# B&R Automation Studio project PLC code - cp (part 20)

#### Kernel2PLC_AutoCode.st
```iecst
// THIS CODE IS AUTOGENERATED. DO NOT MODIFY IT WITH AUTOMATION STUDIO
// Generation: 10/07/2024 16:17:34
// Program version: 2.1.4.0

ACTION Kernel2PLC_AutoCode:
gMachine.parSw.Clean.tiBetweenCleaningBlocks:=SECONDS_TO_TIME(HoldingRegister[3000]*1);
gMachine.parSw.Clean.iCleaningType:=HoldingRegister[3001];
gDing.parSw.rCalibrationValue:=INT_TO_REAL(HoldingRegister[3002])/10;
gMachine.parSw.Media.rThickness:=INT_TO_REAL(HoldingRegister[3003])/10;
gInks[1].parSw.NegPump.rLimitMeniscusDiffWarning:=INT_TO_REAL(HoldingRegister[3004])/10;
gInks[2].parSw.NegPump.rLimitMeniscusDiffWarning:=INT_TO_REAL(HoldingRegister[3005])/10;
gInks[3].parSw.NegPump.rLimitMeniscusDiffWarning:=INT_TO_REAL(HoldingRegister[3006])/10;
gInks[4].parSw.NegPump.rLimitMeniscusDiffWarning:=INT_TO_REAL(HoldingRegister[3007])/10;
gInks[5].parSw.NegPump.rLimitMeniscusDiffWarning:=INT_TO_REAL(HoldingRegister[3008])/10;
gInks[6].parSw.NegPump.rLimitMeniscusDiffWarning:=INT_TO_REAL(HoldingRegister[3009])/10;
gInks[7].parSw.NegPump.rLimitMeniscusDiffWarning:=INT_TO_REAL(HoldingRegister[3010])/10;
gInks[8].parSw.NegPump.rLimitMeniscusDiffWarning:=INT_TO_REAL(HoldingRegister[3011])/10;
gInks[9].parSw.NegPump.rLimitMeniscusDiffWarning:=INT_TO_REAL(HoldingRegister[3012])/10;
gInks[10].parSw.NegPump.rLimitMeniscusDiffWarning:=INT_TO_REAL(HoldingRegister[3013])/10;
gInks[11].parSw.NegPump.rLimitMeniscusDiffWarning:=INT_TO_REAL(HoldingRegister[3014])/10;
gInks[12].parSw.NegPump.rLimitMeniscusDiffWarning:=INT_TO_REAL(HoldingRegister[3015])/10;
gMachine.parSw.rMarginPrint:=INT_TO_REAL(HoldingRegister[3016])/10;
gMachine.parSw.Media.rWidth:=INT_TO_REAL(HoldingRegister[3017])/10;
gNonCrash[1].parSw.rGearBox:=INT_TO_REAL(HoldingRegister[3018])/1;
gNonCrash[1].parSw.rPerimeter:=INT_TO_REAL(HoldingRegister[3019])/10;
gNonCrash[1].parSw.rSpeedOffset:=INT_TO_REAL(HoldingRegister[3020])/10;
gMachine.parSw.rFirstHeadPosition:=INT_TO_REAL(HoldingRegister[3021])/1;
gMachine.parSw.rLastHeadPosition:=INT_TO_REAL(HoldingRegister[3022])/1;
gInks[1].parSw.PosPump.rSetPoint:=INT_TO_REAL(HoldingRegister[3023])/10;
gInks[2].parSw.PosPump.rSetPoint:=INT_TO_REAL(HoldingRegister[3024])/10;
gInks[3].parSw.PosPump.rSetPoint:=INT_TO_REAL(HoldingRegister[3025])/10;
gInks[4].parSw.PosPump.rSetPoint:=INT_TO_REAL(HoldingRegister[3026])/10;
gInks[5].parSw.PosPump.rSetPoint:=INT_TO_REAL(HoldingRegister[3027])/10;
gInks[6].parSw.PosPump.rSetPoint:=INT_TO_REAL(HoldingRegister[3028])/10;
gInks[7].parSw.PosPump.rSetPoint:=INT_TO_REAL(HoldingRegister[3029])/10;
gInks[8].parSw.PosPump.rSetPoint:=INT_TO_REAL(HoldingRegister[3030])/10;
gInks[9].parSw.PosPump.rSetPoint:=INT_TO_REAL(HoldingRegister[3031])/10;
gInks[10].parSw.PosPump.rSetPoint:=INT_TO_REAL(HoldingRegister[3032])/10;
gInks[11].parSw.PosPump.rSetPoint:=INT_TO_REAL(HoldingRegister[3033])/10;
gInks[12].parSw.PosPump.rSetPoint:=INT_TO_REAL(HoldingRegister[3034])/10;
gInks[1].parSw.NegPump.rSetPointMeniscus:=INT_TO_REAL(HoldingRegister[3035])/1;
gInks[2].parSw.NegPump.rSetPointMeniscus:=INT_TO_REAL(HoldingRegister[3036])/1;
gInks[3].parSw.NegPump.rSetPointMeniscus:=INT_TO_REAL(HoldingRegister[3037])/1;
gInks[4].parSw.NegPump.rSetPointMeniscus:=INT_TO_REAL(HoldingRegister[3038])/1;
gInks[5].parSw.NegPump.rSetPointMeniscus:=INT_TO_REAL(HoldingRegister[3039])/1;
gInks[6].parSw.NegPump.rSetPointMeniscus:=INT_TO_REAL(HoldingRegister[3040])/1;
gInks[7].parSw.NegPump.rSetPointMeniscus:=INT_TO_REAL(HoldingRegister[3041])/1;
gInks[8].parSw.NegPump.rSetPointMeniscus:=INT_TO_REAL(HoldingRegister[3042])/1;
gInks[9].parSw.NegPump.rSetPointMeniscus:=INT_TO_REAL(HoldingRegister[3043])/1;
gInks[10].parSw.NegPump.rSetPointMeniscus:=INT_TO_REAL(HoldingRegister[3044])/1;
gInks[11].parSw.NegPump.rSetPointMeniscus:=INT_TO_REAL(HoldingRegister[3045])/1;
gInks[12].parSw.NegPump.rSetPointMeniscus:=INT_TO_REAL(HoldingRegister[3046])/1;
gInks[1].parSw.Temp.rSetPointTemp:=INT_TO_REAL(HoldingRegister[3047])/10;
gInks[2].parSw.Temp.rSetPointTemp:=INT_TO_REAL(HoldingRegister[3048])/10;
gInks[3].parSw.Temp.rSetPointTemp:=INT_TO_REAL(HoldingRegister[3049])/10;
gInks[4].parSw.Temp.rSetPointTemp:=INT_TO_REAL(HoldingRegister[3050])/10;
gInks[5].parSw.Temp.rSetPointTemp:=INT_TO_REAL(HoldingRegister[3051])/10;
gInks[6].parSw.Temp.rSetPointTemp:=INT_TO_REAL(HoldingRegister[3052])/10;
gInks[7].parSw.Temp.rSetPointTemp:=INT_TO_REAL(HoldingRegister[3053])/10;
gInks[8].parSw.Temp.rSetPointTemp:=INT_TO_REAL(HoldingRegister[3054])/10;
gInks[9].parSw.Temp.rSetPointTemp:=INT_TO_REAL(HoldingRegister[3055])/10;
gInks[10].parSw.Temp.rSetPointTemp:=INT_TO_REAL(HoldingRegister[3056])/10;
gInks[11].parSw.Temp.rSetPointTemp:=INT_TO_REAL(HoldingRegister[3057])/10;
gInks[12].parSw.Temp.rSetPointTemp:=INT_TO_REAL(HoldingRegister[3058])/10;
gMachine.parSw.rBeltSpeedSetPoint:=INT_TO_REAL(HoldingRegister[3071])/10;
gInks[1].parSw.NegPump.rSetPointManual:=INT_TO_REAL(HoldingRegister[3072])/10;
gInks[2].parSw.NegPump.rSetPointManual:=INT_TO_REAL(HoldingRegister[3073])/10;
gInks[3].parSw.NegPump.rSetPointManual:=INT_TO_REAL(HoldingRegister[3074])/10;
gInks[4].parSw.NegPump.rSetPointManual:=INT_TO_REAL(HoldingRegister[3075])/10;
gInks[5].parSw.NegPump.rSetPointManual:=INT_TO_REAL(HoldingRegister[3076])/10;
gInks[6].parSw.NegPump.rSetPointManual:=INT_TO_REAL(HoldingRegister[3077])/10;
gInks[7].parSw.NegPump.rSetPointManual:=INT_TO_REAL(HoldingRegister[3078])/10;
gInks[8].parSw.NegPump.rSetPointManual:=INT_TO_REAL(HoldingRegister[3079])/10;
gInks[9].parSw.NegPump.rSetPointManual:=INT_TO_REAL(HoldingRegister[3080])/10;
gInks[10].parSw.NegPump.rSetPointManual:=INT_TO_REAL(HoldingRegister[3081])/10;
gInks[11].parSw.NegPump.rSetPointManual:=INT_TO_REAL(HoldingRegister[3082])/10;
gInks[12].parSw.NegPump.rSetPointManual:=INT_TO_REAL(HoldingRegister[3083])/10;
gInks[1].parSw.PosPump.rSetPointManual:=INT_TO_REAL(HoldingRegister[3084])/1;
gInks[2].parSw.PosPump.rSetPointManual:=INT_TO_REAL(HoldingRegister[3085])/1;
gInks[3].parSw.PosPump.rSetPointManual:=INT_TO_REAL(HoldingRegister[3086])/1;
gInks[4].parSw.PosPump.rSetPointManual:=INT_TO_REAL(HoldingRegister[3087])/1;
gInks[5].parSw.PosPump.rSetPointManual:=INT_TO_REAL(HoldingRegister[3088])/1;
gInks[6].parSw.PosPump.rSetPointManual:=INT_TO_REAL(HoldingRegister[3089])/1;
gInks[7].parSw.PosPump.rSetPointManual:=INT_TO_REAL(HoldingRegister[3090])/1;
gInks[8].parSw.PosPump.rSetPointManual:=INT_TO_REAL(HoldingRegister[3091])/1;
gInks[9].parSw.PosPump.rSetPointManual:=INT_TO_REAL(HoldingRegister[3092])/1;
gInks[10].parSw.PosPump.rSetPointManual:=INT_TO_REAL(HoldingRegister[3093])/1;
gInks[11].parSw.PosPump.rSetPointManual:=INT_TO_REAL(HoldingRegister[3094])/1;
gInks[12].parSw.PosPump.rSetPointManual:=INT_TO_REAL(HoldingRegister[3095])/1;
gMachine.parSw.tiDelayConsent:=SECONDS_TO_TIME(HoldingRegister[3096]*1);
gPhotoCells.parSw.rThicknessReference:=INT_TO_REAL(HoldingRegister[3097])/10;
gMachine.parSw.Clean.tiToCleanWhenPrinterStopped:=MINUTES_TO_TIME(HoldingRegister[3098]*1);
gTime.Params.UTCTimeZone:=HoldingRegister[3099];
gMachine.parSw.Clean.iCleanMotorSpeedFwd:=HoldingRegister[3100];
gMachine.parSw.Clean.iCleanMotorSpeedBwd:=HoldingRegister[3101];
ComandBool(In:=gMachine.parSw.Hw.xInstallnSensor,Com:=HoldingRegister[4000]);
ComandBool(In:=gTransVacuum[1].parSw.xActiveOutOfProduction,Com:=HoldingRegister[4001]);
ComandBool(In:=gTransVacuum[1].OrdersSw.xRunManual,Com:=HoldingRegister[4002]);
ComandBool(In:=gInks[1].parSw.xActTestMode,Com:=HoldingRegister[4003]);
ComandBool(In:=gInks[2].parSw.xActTestMode,Com:=HoldingRegister[4004]);
ComandBool(In:=gInks[3].parSw.xActTestMode,Com:=HoldingRegister[4005]);
ComandBool(In:=gInks[4].parSw.xActTestMode,Com:=HoldingRegister[4006]);
ComandBool(In:=gInks[5].parSw.xActTestMode,Com:=HoldingRegister[4007]);
ComandBool(In:=gInks[6].parSw.xActTestMode,Com:=HoldingRegister[4008]);
ComandBool(In:=gInks[7].parSw.xActTestMode,Com:=HoldingRegister[4009]);
ComandBool(In:=gInks[8].parSw.xActTestMode,Com:=HoldingRegister[4010]);
ComandBool(In:=gInks[9].parSw.xActTestMode,Com:=HoldingRegister[4011]);
ComandBool(In:=gInks[10].parSw.xActTestMode,Com:=HoldingRegister[4012]);
ComandBool(In:=gInks[11].parSw.xActTestMode,Com:=HoldingRegister[4013]);
ComandBool(In:=gInks[12].parSw.xActTestMode,Com:=HoldingRegister[4014]);
ComandBool(In:=gInks[1].parSw.xEnabledBarToPrint,Com:=HoldingRegister[4015]);
ComandBool(In:=gInks[2].parSw.xEnabledBarToPrint,Com:=HoldingRegister[4016]);
ComandBool(In:=gInks[3].parSw.xEnabledBarToPrint,Com:=HoldingRegister[4017]);
ComandBool(In:=gInks[4].parSw.xEnabledBarToPrint,Com:=HoldingRegister[4018]);
ComandBool(In:=gInks[5].parSw.xEnabledBarToPrint,Com:=HoldingRegister[4019]);
ComandBool(In:=gInks[6].parSw.xEnabledBarToPrint,Com:=HoldingRegister[4020]);
ComandBool(In:=gInks[7].parSw.xEnabledBarToPrint,Com:=HoldingRegister[4021]);
ComandBool(In:=gInks[8].parSw.xEnabledBarToPrint,Com:=HoldingRegister[4022]);
ComandBool(In:=gInks[9].parSw.xEnabledBarToPrint,Com:=HoldingRegister[4023]);
ComandBool(In:=gInks[10].parSw.xEnabledBarToPrint,Com:=HoldingRegister[4024]);
ComandBool(In:=gInks[11].parSw.xEnabledBarToPrint,Com:=HoldingRegister[4025]);
ComandBool(In:=gInks[12].parSw.xEnabledBarToPrint,Com:=HoldingRegister[4026]);
gTransVacuum[1].parSw.rVacPressureSetPointPerc:=INT_TO_REAL(HoldingRegister[4027])/10;
ComandBool(In:=gMachine.commandsSw.xToByPass_GI,Com:=HoldingRegister[4028]);
gMachine.parSw.Clean.iPiecesNumberToCleanL1:=HoldingRegister[4029];
gMachine.parSw.Clean.iPiecesNumberToCleanL2:=HoldingRegister[4030];
ComandBool(In:=gBlock[1].commands.xForceCleanNoDelay,Com:=HoldingRegister[4031]);
ComandBool(In:=gBlock[2].commands.xForceCleanNoDelay,Com:=HoldingRegister[4032]);
ComandBool(In:=gMachine.parSw.Clean.xCleaningBlocksInSeq,Com:=HoldingRegister[4033]);
gMachine.parSw.Safety.rMountedPieceOverthickness:=INT_TO_REAL(HoldingRegister[4036])/10;
ComandBool(In:=gMachine.parSw.Shot.xShotLine1,Com:=HoldingRegister[4038]);
ComandBool(In:=gMachine.parSw.Shot.xShotLine2,Com:=HoldingRegister[4039]);
ComandBool(In:=gMachine.parSw.Dtp.xDoubleLine,Com:=HoldingRegister[4040]);
gMachine.parSw.CleanBelt.tiCleaningBeltDuration:=SECONDS_TO_TIME(HoldingRegister[4041]*1);
gMachine.parSw.CleanBeltTop.tiCleaningBeltDuration:=SECONDS_TO_TIME(HoldingRegister[4042]*1);
ComandBool(In:=gBlock[1].commands.xEnableCleaningWithWater,Com:=HoldingRegister[4043]);
ComandBool(In:=gBlock[2].commands.xEnableCleaningWithWater,Com:=HoldingRegister[4044]);
ComandBool(In:=gMachine.parSw.xJamDetectEnable,Com:=HoldingRegister[4046]);
ComandBool(In:=gMachine.parSw.Clean.xEnableCleaningInStopMode,Com:=HoldingRegister[4047]);
ComandBool(In:=gBlock[1].parSw.xEnableToMovements,Com:=HoldingRegister[4048]);
ComandBool(In:=gBlock[2].parSw.xEnableToMovements,Com:=HoldingRegister[4049]);
ComandBool(In:=gNonCrash[1].parSw.xEnable,Com:=HoldingRegister[4050]);
ComandBool(In:=gInks[1].parSw.Temp.xTankHeaterEnabled,Com:=HoldingRegister[4051]);
ComandBool(In:=gInks[2].parSw.Temp.xTankHeaterEnabled,Com:=HoldingRegister[4052]);
ComandBool(In:=gInks[3].parSw.Temp.xTankHeaterEnabled,Com:=HoldingRegister[4053]);
ComandBool(In:=gInks[4].parSw.Temp.xTankHeaterEnabled,Com:=HoldingRegister[4054]);
ComandBool(In:=gInks[5].parSw.Temp.xTankHeaterEnabled,Com:=HoldingRegister[4055]);
ComandBool(In:=gInks[6].parSw.Temp.xTankHeaterEnabled,Com:=HoldingRegister[4056]);
ComandBool(In:=gInks[7].parSw.Temp.xTankHeaterEnabled,Com:=HoldingRegister[4057]);
ComandBool(In:=gInks[8].parSw.Temp.xTankHeaterEnabled,Com:=HoldingRegister[4058]);
ComandBool(In:=gInks[9].parSw.Temp.xTankHeaterEnabled,Com:=HoldingRegister[4059]);
ComandBool(In:=gInks[10].parSw.Temp.xTankHeaterEnabled,Com:=HoldingRegister[4060]);
ComandBool(In:=gInks[11].parSw.Temp.xTankHeaterEnabled,Com:=HoldingRegister[4061]);
ComandBool(In:=gInks[12].parSw.Temp.xTankHeaterEnabled,Com:=HoldingRegister[4062]);
ComandBool(In:=gBlock[1].parSw.xEnableToPrint,Com:=HoldingRegister[4063]);
ComandBool(In:=gBlock[2].parSw.xEnableToPrint,Com:=HoldingRegister[4064]);
ComandBool(In:=gMachine.parSw.Electronics.xPrintServerOK,Com:=HoldingRegister[4065]);
ComandBool(In:=gMachine.parSw.Electronics.xRobotReadyL1,Com:=HoldingRegister[4066]);
ComandBool(In:=gMachine.parSw.Electronics.xRobotReadyL2,Com:=HoldingRegister[4067]);
ComandBool(In:=gMachine.parSw.PCs.xExistPC1,Com:=HoldingRegister[4068]);
ComandBool(In:=gMachine.parSw.PCs.xExistPC2,Com:=HoldingRegister[4069]);
gMachine.parSw.iFaultComPcPlc:=HoldingRegister[4070];
ComandBool(In:=gBlock[1].commands.xForceCleanDelay,Com:=HoldingRegister[4073]);
ComandBool(In:=gBlock[2].commands.xForceCleanDelay,Com:=HoldingRegister[4074]);
ComandBool(In:=gBlock[1].commands.xToCleanPosition,Com:=HoldingRegister[4075]);
ComandBool(In:=gBlock[2].commands.xToCleanPosition,Com:=HoldingRegister[4076]);
ComandBool(In:=gMachine.parSw.CleanBelt.xCleanBeltByTiles,Com:=HoldingRegister[4077]);
ComandBool(In:=gMachine.parSw.CleanBelt.xCleanBeltByTime,Com:=HoldingRegister[4078]);
ComandBool(In:=gMachine.parSw.CleanBeltTop.xCleanBeltByTiles,Com:=HoldingRegister[4079]);
ComandBool(In:=gMachine.parSw.CleanBeltTop.xCleanBeltByTime,Com:=HoldingRegister[4080]);
ComandBool(In:=gBlock[1].commands.Manual.xManIclaBack,Com:=HoldingRegister[4081]);
ComandBool(In:=gBlock[2].commands.Manual.xManIclaBack,Com:=HoldingRegister[4082]);
ComandBool(In:=gBlock[1].commands.Manual.xManBarsDown,Com:=HoldingRegister[4083]);
ComandBool(In:=gBlock[2].commands.Manual.xManBarsDown,Com:=HoldingRegister[4084]);
ComandBool(In:=gBlock[1].commands.Manual.xManIclaForward,Com:=HoldingRegister[4085]);
ComandBool(In:=gBlock[2].commands.Manual.xManIclaForward,Com:=HoldingRegister[4086]);
gInks[1].parSw.iInkConsumption:=HoldingRegister[4087];
gInks[2].parSw.iInkConsumption:=HoldingRegister[4088];
gInks[3].parSw.iInkConsumption:=HoldingRegister[4089];
gInks[4].parSw.iInkConsumption:=HoldingRegister[4090];
gInks[5].parSw.iInkConsumption:=HoldingRegister[4091];
gInks[6].parSw.iInkConsumption:=HoldingRegister[4092];
gInks[7].parSw.iInkConsumption:=HoldingRegister[4093];
gInks[8].parSw.iInkConsumption:=HoldingRegister[4094];
gInks[9].parSw.iInkConsumption:=HoldingRegister[4095];
gInks[10].parSw.iInkConsumption:=HoldingRegister[4096];
gInks[11].parSw.iInkConsumption:=HoldingRegister[4097];
gInks[12].parSw.iInkConsumption:=HoldingRegister[4098];
ComandBool(In:=gInks[1].parSw.xReverseOnManual,Com:=HoldingRegister[4099]);
ComandBool(In:=gInks[2].parSw.xReverseOnManual,Com:=HoldingRegister[4100]);
ComandBool(In:=gInks[3].parSw.xReverseOnManual,Com:=HoldingRegister[4101]);
ComandBool(In:=gInks[4].parSw.xReverseOnManual,Com:=HoldingRegister[4102]);
ComandBool(In:=gInks[5].parSw.xReverseOnManual,Com:=HoldingRegister[4103]);
ComandBool(In:=gInks[6].parSw.xReverseOnManual,Com:=HoldingRegister[4104]);
ComandBool(In:=gInks[7].parSw.xReverseOnManual,Com:=HoldingRegister[4105]);
ComandBool(In:=gInks[8].parSw.xReverseOnManual,Com:=HoldingRegister[4106]);
ComandBool(In:=gInks[9].parSw.xReverseOnManual,Com:=HoldingRegister[4107]);
ComandBool(In:=gInks[10].parSw.xReverseOnManual,Com:=HoldingRegister[4108]);
ComandBool(In:=gInks[11].parSw.xReverseOnManual,Com:=HoldingRegister[4109]);
ComandBool(In:=gInks[12].parSw.xReverseOnManual,Com:=HoldingRegister[4110]);
gInks[1].parSw.Config.iInkType:=HoldingRegister[4111];
gInks[2].parSw.Config.iInkType:=HoldingRegister[4112];
gInks[3].parSw.Config.iInkType:=HoldingRegister[4113];
gInks[4].parSw.Config.iInkType:=HoldingRegister[4114];
gInks[5].parSw.Config.iInkType:=HoldingRegister[4115];
gInks[6].parSw.Config.iInkType:=HoldingRegister[4116];
gInks[7].parSw.Config.iInkType:=HoldingRegister[4117];
gInks[8].parSw.Config.iInkType:=HoldingRegister[4118];
gInks[9].parSw.Config.iInkType:=HoldingRegister[4119];
gInks[10].parSw.Config.iInkType:=HoldingRegister[4120];
gInks[11].parSw.Config.iInkType:=HoldingRegister[4121];
gInks[12].parSw.Config.iInkType:=HoldingRegister[4122];
ComandBool(In:=gMachine.commandsSw.xStart_GI,Com:=HoldingRegister[4123]);
ComandBool(In:=gMachine.commandsSw.xStop_GI,Com:=HoldingRegister[4124]);
ComandBool(In:=gMachine.commandsSw.xPause_GI,Com:=HoldingRegister[4125]);
ComandBool(In:=gMachine.commands.xCompenserLine1,Com:=HoldingRegister[4126]);
ComandBool(In:=gMachine.commands.xCompenserLine2,Com:=HoldingRegister[4127]);
ComandBool(In:=gBlock[1].commands.Manual.xManBarsUp,Com:=HoldingRegister[4128]);
ComandBool(In:=gBlock[2].commands.Manual.xManBarsUp,Com:=HoldingRegister[4129]);
ComandBool(In:=gBlock[1].commands.xIclaHomeOrderInterrupt,Com:=HoldingRegister[4130]);
ComandBool(In:=gBlock[2].commands.xIclaHomeOrderInterrupt,Com:=HoldingRegister[4131]);
ComandBool(In:=gMachine.parSw.Electronics.xIsPBF,Com:=HoldingRegister[4132]);
ComandBool(In:=gMachine.commandsSw.xToLaboratory_GI,Com:=HoldingRegister[4133]);
gMachine.parSw.CleanBelt.iSPTilesToCleanBelt:=HoldingRegister[4134];
ComandBool(In:=gMachine.parSw.CleanBelt.xCleanBeltContinue,Com:=HoldingRegister[4135]);
gMachine.parSw.CleanBeltTop.iSPTilesToCleanBelt:=HoldingRegister[4136];
ComandBool(In:=gMachine.parSw.CleanBeltTop.xCleanBeltContinue,Com:=HoldingRegister[4137]);
ComandBool(In:=gInks[1].ordersSw.xStartManual,Com:=HoldingRegister[4138]);
ComandBool(In:=gInks[2].ordersSw.xStartManual,Com:=HoldingRegister[4139]);
ComandBool(In:=gInks[3].ordersSw.xStartManual,Com:=HoldingRegister[4140]);
ComandBool(In:=gInks[4].ordersSw.xStartManual,Com:=HoldingRegister[4141]);
ComandBool(In:=gInks[5].ordersSw.xStartManual,Com:=HoldingRegister[4142]);
ComandBool(In:=gInks[6].ordersSw.xStartManual,Com:=HoldingRegister[4143]);
ComandBool(In:=gInks[7].ordersSw.xStartManual,Com:=HoldingRegister[4144]);
ComandBool(In:=gInks[8].ordersSw.xStartManual,Com:=HoldingRegister[4145]);
ComandBool(In:=gInks[9].ordersSw.xStartManual,Com:=HoldingRegister[4146]);
ComandBool(In:=gInks[10].ordersSw.xStartManual,Com:=HoldingRegister[4147]);
ComandBool(In:=gInks[11].ordersSw.xStartManual,Com:=HoldingRegister[4148]);
ComandBool(In:=gInks[12].ordersSw.xStartManual,Com:=HoldingRegister[4149]);
ComandBool(In:=gMachine.parSw.CleanBelt.xCleanBeltForced,Com:=HoldingRegister[4150]);
ComandBool(In:=gMachine.parSw.CleanBeltTop.xCleanBeltForced,Com:=HoldingRegister[4151]);
ComandBool(In:=gMachine.parSw.Clean.xCleanSystemByPieces,Com:=HoldingRegister[4152]);
ComandBool(In:=gMachine.parSw.Clean.xCleanSystemByTime,Com:=HoldingRegister[4153]);
ComandBool(In:=gBlock[1].commands.Manual.xManTrayIn,Com:=HoldingRegister[4154]);
ComandBool(In:=gBlock[2].commands.Manual.xManTrayIn,Com:=HoldingRegister[4155]);
ComandBool(In:=gBlock[1].commands.Manual.xManTrayOut,Com:=HoldingRegister[4156]);
ComandBool(In:=gBlock[2].commands.Manual.xManTrayOut,Com:=HoldingRegister[4157]);
ComandBool(In:=gMachine.parSw.xMachineDirection,Com:=HoldingRegister[4159]);
ComandBool(In:=gMachine.parSw.PCs.xKeepPcsOn,Com:=HoldingRegister[4161]);
gTransVacuum[1].parSw.rManSetPoint:=INT_TO_REAL(HoldingRegister[4162])/10;
ComandBool(In:=gBlock[1].commands.Manual.xManVenturi,Com:=HoldingRegister[4163]);
ComandBool(In:=gBlock[2].commands.Manual.xManVenturi,Com:=HoldingRegister[4164]);
gInks[1].parSw.Config.iMappingBar:=HoldingRegister[4165];
gInks[2].parSw.Config.iMappingBar:=HoldingRegister[4166];
gInks[3].parSw.Config.iMappingBar:=HoldingRegister[4167];
gInks[4].parSw.Config.iMappingBar:=HoldingRegister[4168];
gInks[5].parSw.Config.iMappingBar:=HoldingRegister[4169];
gInks[6].parSw.Config.iMappingBar:=HoldingRegister[4170];
gInks[7].parSw.Config.iMappingBar:=HoldingRegister[4171];
gInks[8].parSw.Config.iMappingBar:=HoldingRegister[4172];
gInks[9].parSw.Config.iMappingBar:=HoldingRegister[4173];
gInks[10].parSw.Config.iMappingBar:=HoldingRegister[4174];
gInks[11].parSw.Config.iMappingBar:=HoldingRegister[4175];
gInks[12].parSw.Config.iMappingBar:=HoldingRegister[4176];
ComandBool(In:=gInks[1].ordersSw.xStartInks,Com:=HoldingRegister[4177]);
ComandBool(In:=gInks[2].ordersSw.xStartInks,Com:=HoldingRegister[4178]);
ComandBool(In:=gInks[3].ordersSw.xStartInks,Com:=HoldingRegister[4179]);
ComandBool(In:=gInks[4].ordersSw.xStartInks,Com:=HoldingRegister[4180]);
ComandBool(In:=gInks[5].ordersSw.xStartInks,Com:=HoldingRegister[4181]);
ComandBool(In:=gInks[6].ordersSw.xStartInks,Com:=HoldingRegister[4182]);
ComandBool(In:=gInks[7].ordersSw.xStartInks,Com:=HoldingRegister[4183]);
ComandBool(In:=gInks[8].ordersSw.xStartInks,Com:=HoldingRegister[4184]);
ComandBool(In:=gInks[9].ordersSw.xStartInks,Com:=HoldingRegister[4185]);
ComandBool(In:=gInks[10].ordersSw.xStartInks,Com:=HoldingRegister[4186]);
ComandBool(In:=gInks[11].ordersSw.xStartInks,Com:=HoldingRegister[4187]);
ComandBool(In:=gInks[12].ordersSw.xStartInks,Com:=HoldingRegister[4188]);
gMachine.parSw.Safety.rMarginSafePrint:=INT_TO_REAL(HoldingRegister[4189])/10;
gMachine.parSw.Media.rLength:=INT_TO_REAL(HoldingRegister[4190])/10;
gBelt.parSw.rAxisLength:=INT_TO_REAL(HoldingRegister[4191])/10;
gMachine.parSw.Dtp.iModeLine1:=HoldingRegister[4192];
gMachine.parSw.Dtp.iModeLine2:=HoldingRegister[4193];
gMachine.parSw.Suction.iBlowerMode:=HoldingRegister[4194];
ComandBool(In:=gMachine.commandsSw.xToNormal_GI,Com:=HoldingRegister[4195]);
gBlock[1].parSw.rOffsetCleanMtrAdjust:=INT_TO_REAL(HoldingRegister[4196])/10;
gBlock[2].parSw.rOffsetCleanMtrAdjust:=INT_TO_REAL(HoldingRegister[4197])/10;
gBlock[1].parSw.rOffsetCleanMtrOperatr:=INT_TO_REAL(HoldingRegister[4198])/10;
gBlock[2].parSw.rOffsetCleanMtrOperatr:=INT_TO_REAL(HoldingRegister[4199])/10;
ComandBool(In:=gInks[1].parSw.xOnReverseCapped,Com:=HoldingRegister[4200]);
ComandBool(In:=gInks[2].parSw.xOnReverseCapped,Com:=HoldingRegister[4201]);
ComandBool(In:=gInks[3].parSw.xOnReverseCapped,Com:=HoldingRegister[4202]);
ComandBool(In:=gInks[4].parSw.xOnReverseCapped,Com:=HoldingRegister[4203]);
ComandBool(In:=gInks[5].parSw.xOnReverseCapped,Com:=HoldingRegister[4204]);
ComandBool(In:=gInks[6].parSw.xOnReverseCapped,Com:=HoldingRegister[4205]);
ComandBool(In:=gInks[7].parSw.xOnReverseCapped,Com:=HoldingRegister[4206]);
ComandBool(In:=gInks[8].parSw.xOnReverseCapped,Com:=HoldingRegister[4207]);
ComandBool(In:=gInks[9].parSw.xOnReverseCapped,Com:=HoldingRegister[4208]);
ComandBool(In:=gInks[10].parSw.xOnReverseCapped,Com:=HoldingRegister[4209]);
ComandBool(In:=gInks[11].parSw.xOnReverseCapped,Com:=HoldingRegister[4210]);
ComandBool(In:=gInks[12].parSw.xOnReverseCapped,Com:=HoldingRegister[4211]);
ComandBool(In:=gInks[1].parSw.xOnReverseCleaning,Com:=HoldingRegister[4212]);
ComandBool(In:=gInks[2].parSw.xOnReverseCleaning,Com:=HoldingRegister[4213]);
ComandBool(In:=gInks[3].parSw.xOnReverseCleaning,Com:=HoldingRegister[4214]);
ComandBool(In:=gInks[4].parSw.xOnReverseCleaning,Com:=HoldingRegister[4215]);
ComandBool(In:=gInks[5].parSw.xOnReverseCleaning,Com:=HoldingRegister[4216]);
ComandBool(In:=gInks[6].parSw.xOnReverseCleaning,Com:=HoldingRegister[4217]);
ComandBool(In:=gInks[7].parSw.xOnReverseCleaning,Com:=HoldingRegister[4218]);
ComandBool(In:=gInks[8].parSw.xOnReverseCleaning,Com:=HoldingRegister[4219]);
ComandBool(In:=gInks[9].parSw.xOnReverseCleaning,Com:=HoldingRegister[4220]);
ComandBool(In:=gInks[10].parSw.xOnReverseCleaning,Com:=HoldingRegister[4221]);
ComandBool(In:=gInks[11].parSw.xOnReverseCleaning,Com:=HoldingRegister[4222]);
ComandBool(In:=gInks[12].parSw.xOnReverseCleaning,Com:=HoldingRegister[4223]);
ComandBool(In:=gMachine.commands.xAllToCap,Com:=HoldingRegister[4224]);
ComandBool(In:=gMachine.commands.xAllToPrint,Com:=HoldingRegister[4225]);
ComandBool(In:=gPhotoCells.ordersSw.xMoveDown,Com:=HoldingRegister[4226]);
gPhotoCells.parSw.rMechOffset:=INT_TO_REAL(HoldingRegister[4227])/10;
ComandBool(In:=gPhotoCells.ordersSw.xMoveUp,Com:=HoldingRegister[4228]);
ComandBool(In:=gInks[1].ordersSw.xPowPrintHead,Com:=HoldingRegister[4229]);
ComandBool(In:=gInks[2].ordersSw.xPowPrintHead,Com:=HoldingRegister[4230]);
ComandBool(In:=gInks[3].ordersSw.xPowPrintHead,Com:=HoldingRegister[4231]);
ComandBool(In:=gInks[4].ordersSw.xPowPrintHead,Com:=HoldingRegister[4232]);
ComandBool(In:=gInks[5].ordersSw.xPowPrintHead,Com:=HoldingRegister[4233]);
ComandBool(In:=gInks[6].ordersSw.xPowPrintHead,Com:=HoldingRegister[4234]);
ComandBool(In:=gInks[7].ordersSw.xPowPrintHead,Com:=HoldingRegister[4235]);
ComandBool(In:=gInks[8].ordersSw.xPowPrintHead,Com:=HoldingRegister[4236]);
ComandBool(In:=gInks[9].ordersSw.xPowPrintHead,Com:=HoldingRegister[4237]);
ComandBool(In:=gInks[10].ordersSw.xPowPrintHead,Com:=HoldingRegister[4238]);
ComandBool(In:=gInks[11].ordersSw.xPowPrintHead,Com:=HoldingRegister[4239]);
ComandBool(In:=gInks[12].ordersSw.xPowPrintHead,Com:=HoldingRegister[4240]);
gInks[1].parSw.iInkEnabledPrintHeads:=HoldingRegister[4241];
gInks[2].parSw.iInkEnabledPrintHeads:=HoldingRegister[4242];
gInks[3].parSw.iInkEnabledPrintHeads:=HoldingRegister[4243];
gInks[4].parSw.iInkEnabledPrintHeads:=HoldingRegister[4244];
gInks[5].parSw.iInkEnabledPrintHeads:=HoldingRegister[4245];
gInks[6].parSw.iInkEnabledPrintHeads:=HoldingRegister[4246];
gInks[7].parSw.iInkEnabledPrintHeads:=HoldingRegister[4247];
gInks[8].parSw.iInkEnabledPrintHeads:=HoldingRegister[4248];
gInks[9].parSw.iInkEnabledPrintHeads:=HoldingRegister[4249];
gInks[10].parSw.iInkEnabledPrintHeads:=HoldingRegister[4250];
gInks[11].parSw.iInkEnabledPrintHeads:=HoldingRegister[4251];
gInks[12].parSw.iInkEnabledPrintHeads:=HoldingRegister[4252];
ComandBool(In:=gPhotoCells.commandsSw.xReference,Com:=HoldingRegister[4253]);
ComandBool(In:=gDing.Commands.xCalibrateThickness,Com:=HoldingRegister[4266]);
ComandBool(In:=gBlock[1].commands.xIclaHomeOrder,Com:=HoldingRegister[4267]);
ComandBool(In:=gBlock[2].commands.xIclaHomeOrder,Com:=HoldingRegister[4268]);
ComandBool(In:=gBlock[1].commands.xBarHomeOrder,Com:=HoldingRegister[4269]);
ComandBool(In:=gBlock[2].commands.xBarHomeOrder,Com:=HoldingRegister[4270]);
gBelt.parSw.rGearBox:=INT_TO_REAL(HoldingRegister[4271])/100;
ComandBool(In:=gMachine.parSw.Shot.xRepetitionShotLine1,Com:=HoldingRegister[4272]);
ComandBool(In:=gMachine.parSw.Shot.xRepetitionShotLine2,Com:=HoldingRegister[4273]);
ComandBool(In:=gMachine.commands.xResetCB,Com:=HoldingRegister[4274]);
ComandBool(In:=gMachine.commandsSw.xReset_GI,Com:=HoldingRegister[4275]);
ComandBool(In:=gMachine.commands.xResetRouter,Com:=HoldingRegister[4276]);
ComandBool(In:=gMachine.commands.xResetStrobePdDiff,Com:=HoldingRegister[4277]);
ComandBool(In:=gInks[1].ordersSw.xOrderReverseMan,Com:=HoldingRegister[4278]);
ComandBool(In:=gInks[2].ordersSw.xOrderReverseMan,Com:=HoldingRegister[4279]);
ComandBool(In:=gInks[3].ordersSw.xOrderReverseMan,Com:=HoldingRegister[4280]);
ComandBool(In:=gInks[4].ordersSw.xOrderReverseMan,Com:=HoldingRegister[4281]);
ComandBool(In:=gInks[5].ordersSw.xOrderReverseMan,Com:=HoldingRegister[4282]);
ComandBool(In:=gInks[6].ordersSw.xOrderReverseMan,Com:=HoldingRegister[4283]);
ComandBool(In:=gInks[7].ordersSw.xOrderReverseMan,Com:=HoldingRegister[4284]);
ComandBool(In:=gInks[8].ordersSw.xOrderReverseMan,Com:=HoldingRegister[4285]);
ComandBool(In:=gInks[9].ordersSw.xOrderReverseMan,Com:=HoldingRegister[4286]);
ComandBool(In:=gInks[10].ordersSw.xOrderReverseMan,Com:=HoldingRegister[4287]);
ComandBool(In:=gInks[11].ordersSw.xOrderReverseMan,Com:=HoldingRegister[4288]);
ComandBool(In:=gInks[12].ordersSw.xOrderReverseMan,Com:=HoldingRegister[4289]);
ComandBool(In:=gBlock[1].commands.Manual.xManWaterSpurt,Com:=HoldingRegister[4290]);
ComandBool(In:=gMachine.commandsSw.xMute_GI,Com:=HoldingRegister[4291]);
ComandBool(In:=gMachine.commandsSw.xToStop_GI,Com:=HoldingRegister[4293]);
gMachine.parSw.Shot.tiShotL1:=MILLISECONDS_TO_TIME(HoldingRegister[4294]*1);
gMachine.parSw.Shot.tiShotL2:=MILLISECONDS_TO_TIME(HoldingRegister[4295]*1);
ComandBool(In:=gChiller[1].parSw.xEnable,Com:=HoldingRegister[4296]);
gMachine.parSw.CleanBelt.tiCleaningBeltByTime:=MINUTES_TO_TIME(HoldingRegister[4297]*1);
gMachine.parSw.CleanBeltTop.tiCleaningBeltByTime:=MINUTES_TO_TIME(HoldingRegister[4298]*1);
gMachine.parSw.Clean.tiCleaningByTime:=MINUTES_TO_TIME(HoldingRegister[4299]*1);
gMachine.parSw.Suction.tiBlowerDelayOff:=MINUTES_TO_TIME(HoldingRegister[4300]*1);
ComandBool(In:=gTime.Params.DayLightSavingsTime,Com:=HoldingRegister[4301]);
gInks[1].parSw.Config.iPrintHeadType:=HoldingRegister[4302];
gInks[2].parSw.Config.iPrintHeadType:=HoldingRegister[4303];
gInks[3].parSw.Config.iPrintHeadType:=HoldingRegister[4304];
gInks[4].parSw.Config.iPrintHeadType:=HoldingRegister[4305];
gInks[5].parSw.Config.iPrintHeadType:=HoldingRegister[4306];
gInks[6].parSw.Config.iPrintHeadType:=HoldingRegister[4307];
gInks[7].parSw.Config.iPrintHeadType:=HoldingRegister[4308];
gInks[8].parSw.Config.iPrintHeadType:=HoldingRegister[4309];
gInks[9].parSw.Config.iPrintHeadType:=HoldingRegister[4310];
gInks[10].parSw.Config.iPrintHeadType:=HoldingRegister[4311];
gInks[11].parSw.Config.iPrintHeadType:=HoldingRegister[4312];
gInks[12].parSw.Config.iPrintHeadType:=HoldingRegister[4313];
gInks[1].parSw.tiDripTime:=MILLISECONDS_TO_TIME(HoldingRegister[4314]*1);
gInks[2].parSw.tiDripTime:=MILLISECONDS_TO_TIME(HoldingRegister[4315]*1);
gInks[3].parSw.tiDripTime:=MILLISECONDS_TO_TIME(HoldingRegister[4316]*1);
gInks[4].parSw.tiDripTime:=MILLISECONDS_TO_TIME(HoldingRegister[4317]*1);
gInks[5].parSw.tiDripTime:=MILLISECONDS_TO_TIME(HoldingRegister[4318]*1);
gInks[6].parSw.tiDripTime:=MILLISECONDS_TO_TIME(HoldingRegister[4319]*1);
gInks[7].parSw.tiDripTime:=MILLISECONDS_TO_TIME(HoldingRegister[4320]*1);
gInks[8].parSw.tiDripTime:=MILLISECONDS_TO_TIME(HoldingRegister[4321]*1);
gInks[9].parSw.tiDripTime:=MILLISECONDS_TO_TIME(HoldingRegister[4322]*1);
gInks[10].parSw.tiDripTime:=MILLISECONDS_TO_TIME(HoldingRegister[4323]*1);
gInks[11].parSw.tiDripTime:=MILLISECONDS_TO_TIME(HoldingRegister[4324]*1);
gInks[12].parSw.tiDripTime:=MILLISECONDS_TO_TIME(HoldingRegister[4325]*1);
gInks[1].parSw.tiReverseManual:=SECONDS_TO_TIME(HoldingRegister[4326]*1);
gInks[2].parSw.tiReverseManual:=SECONDS_TO_TIME(HoldingRegister[4327]*1);
gInks[3].parSw.tiReverseManual:=SECONDS_TO_TIME(HoldingRegister[4328]*1);
gInks[4].parSw.tiReverseManual:=SECONDS_TO_TIME(HoldingRegister[4329]*1);
gInks[5].parSw.tiReverseManual:=SECONDS_TO_TIME(HoldingRegister[4330]*1);
gInks[6].parSw.tiReverseManual:=SECONDS_TO_TIME(HoldingRegister[4331]*1);
gInks[7].parSw.tiReverseManual:=SECONDS_TO_TIME(HoldingRegister[4332]*1);
gInks[8].parSw.tiReverseManual:=SECONDS_TO_TIME(HoldingRegister[4333]*1);
gInks[9].parSw.tiReverseManual:=SECONDS_TO_TIME(HoldingRegister[4334]*1);
gInks[10].parSw.tiReverseManual:=SECONDS_TO_TIME(HoldingRegister[4335]*1);
gInks[11].parSw.tiReverseManual:=SECONDS_TO_TIME(HoldingRegister[4336]*1);
gInks[12].parSw.tiReverseManual:=SECONDS_TO_TIME(HoldingRegister[4337]*1);
gMachine.parSw.Clean.tiTimeDelayToCleanL1:=SECONDS_TO_TIME(HoldingRegister[4338]*1);
gMachine.parSw.Clean.tiTimeDelayToCleanL2:=SECONDS_TO_TIME(HoldingRegister[4339]*1);
gMachine.parSw.Clean.tiTimeDelayGapToClean:=SECONDS_TO_TIME(HoldingRegister[4340]*1);
gTransVacuum[1].parSw.ValvMask:=UDINTFromComms(4342,ADR(HoldingRegister));
ComandBool(In:=gMachine.commands.SerialNumber.xExecute,Com:=HoldingRegister[949]);
END_ACTION
```

#### ReadSerialName.st
```iecst
ACTION ReadSerialName:

	strSerialName ACCESS ADR(HoldingRegister[SERIAL_NAME_ASSIGNATION_ADR]);

	IF brsstrlen(ADR(gMachine.St.HwData.SerialNumber)) <= 4 AND  brsstrlen(ADR(strSerialName)) > 0 THEN
		gMachine.commands.SerialNumber.SerialNumber := strSerialName;
		IF EDGEPOS(HoldingRegister[SERIAL_NAME_TRIGGER_ADR]>0) THEN
			gMachine.commands.SerialNumber.xExecute := TRUE;
			HoldingRegister[SERIAL_NAME_TRIGGER_ADR] := 0;
		END_IF
	END_IF

END_ACTION
```

#### Kernel2PLC.var
```iecst
VAR
	strSerialName : REFERENCE TO STRING[80];
END_VAR
```

### Program Logical/Printer/Comms/PLC2Kernel (IEC)

#### PLC2Kernel.st - Init, cyclic, exit code
```iecst
PROGRAM _CYCLIC

	IF NOT xStarted THEN
		xStarted:=TRUE;
		RETURN;
	END_IF

	//If in Simulation and running without Kernel, do not execute communications
	IF gMachine.St.HwData.Family = FAMILY_BRAUTOMATIONRUNTIME AND (NOT gSimMachine.Parameters.xRunWithKernel OR gMachine.Pt.CommsType=NoCommsType)  THEN
		RETURN;
	END_IF

	//Manual cleaning the RegisterArray
	IF (gMachine.Pt.CommsType=Type_ModbusTcp) AND (xClenanCommsArray OR gMachine.AutoCmd.xCleanModbus) THEN
		FOR iIndexCommsArray:=0 TO 8999 DO
			HoldingRegister[iIndexCommsArray]:=0;
		END_FOR;
		xClenanCommsArray:=FALSE;
		gMachine.AutoCmd.xCleanModbus := FALSE;
	END_IF

	//////////////////////////////////////////////////////////////////////////////////////////////////////////////////
	// COMS   COMS   COMS   COMS   COMS   COMS   COMS   COMS   COMS   COMS   COMS   COMS   COMS   COMS   COMS   COMS
	// COMS   COMS   COMS   COMS   COMS   COMS   COMS   COMS   COMS   COMS   COMS   COMS   COMS   COMS   COMS   COMS
	//////////////////////////////////////////////////////////////////////////////////////////////////////////////////

	//AlarmKernelPLCComms;

	IF gMachine.Pt.CommsType=Type_ModbusTcp THEN
		PLC2Kernel_AutoCode;
	END_IF

	WriteSerialName;

END_PROGRAM
```
